(* IEC 61131-3 sources: ae-simplified-sorting-machine/AX/src/controlModules, 7 files *)

(* ---- IElevator.st ---- *)
NAMESPACE ControlModules

    /// Interface for elevator classes that extends ITransportDevice to add additional
    /// commands relevant for elevator operation
    INTERFACE IElevator extends ITransportDevice
        //=============================================================================
        //SIEMENS AG
        //(c)Copyright 2025 All Rights Reserved
        //-----------------------------------------------------------------------------
        //Tested with:   S7-1500 FW V4.0
        //Engineering:   SIMATIC AX Logic Control Engineering
        //Requirements:  none
        //Functionality: Interface for Transport Devices used as elevators
        //-----------------------------------------------------------------------------
        //Change log table:
        //Version  Date       Expert in charge                Changes applied
        //01.00.00 28.11.2025 Siemens Industry Online Support First Release
        //=============================================================================

        /// Commands the elevator to move upward continuously until upper limit is reached
        /// Enables movement without a specific target position
        METHOD  MoveUp
            VAR_INPUT
                /// Velocity for upward movement
                velocity : INT;
            END_VAR
        END_METHOD

        /// Commands the elevator to move downward continuously until lower limit is reached
        /// Enables movement without a specific target position
        METHOD  MoveDown
            VAR_INPUT
                /// Velocity for downward movement
                velocity : INT;
            END_VAR
        END_METHOD
    END_INTERFACE

END_NAMESPACE

(* ---- ITransportDevice.st ---- *)
NAMESPACE ControlModules

    /// Interface for Transport device Classes.
    INTERFACE ITransportDevice
        //=============================================================================
        //SIEMENS AG
        //(c)Copyright 2025 All Rights Reserved
        //-----------------------------------------------------------------------------
        //Tested with:   S7-1500 FW V4.0
        //Engineering:   SIMATIC AX Logic Control Engineering
        //Requirements:  none
        //Functionality: Interface used for control modules implemented as transport devices
        //-----------------------------------------------------------------------------
        //Change log table:
        //Version  Date       Expert in charge                Changes applied
        //01.00.00 28.11.2025 Siemens Industry Online Support First Release
        //=============================================================================

        /// Enables the transport device for operation
        /// Sets the internal enable flag to allow movement commands
        METHOD Enable
        END_METHOD

        /// Disables the transport device for operation
        /// Sets the internal enable flag to disable movement commands
        METHOD  Disable
        END_METHOD

        /// Stops the transport device operation
        /// Disables the device by setting the enable flag to FALSE
        METHOD  Stop
        END_METHOD

        /// Acknowledges errors on the transport device
        /// Sets the internal error acknowledgment flag to clear error conditions
        METHOD  AckError
        END_METHOD

        /// Gets the enable status of the transport device.
        /// TRUE if device is enabled, FALSE otherwise
        METHOD  GetIsEnabled : BOOL
        END_METHOD

        /// Gets the feedback status of the transport device.
        /// TRUE if movement is done, FALSE otherwise
        METHOD  GetIsDone : BOOL
        END_METHOD

        /// Gets the actual position of the transport device.
        /// Actual position in INT
        METHOD  GetActualPosition : INT
        END_METHOD

        /// Commands the transport device to move to a specified position.
        /// TRUE if movement command was accepted (device enabled), FALSE otherwise
        METHOD  PosAbsolute : BOOL
            VAR_INPUT
                /// Target position for the movement command
                targetPos : INT;
                /// Velocity for the movement (optional)
                velocity : INT := INT#0;
            END_VAR
        END_METHOD

        /// Moves the drive at a specified constant velocity.
        /// Sets the drive to jog mode and starts continuous movement.
        /// TRUE if movement command was accepted (device enabled), FALSE otherwise
        METHOD MoveVelocity : BOOL
            VAR_INPUT
                /// Velocity in LU (Length Units) for the drive
                velocity    : INT;
            END_VAR
        END_METHOD

        /// Executes a relative positioning movement.
        /// Moves the drive by a specified increment from current position.
        /// TRUE if movement command was accepted (device enabled), FALSE otherwise
        METHOD PosRelative : BOOL
            VAR_INPUT
                /// Position increment in LU to move relative to current position
                posIncrement   : INT;
                /// Velocity for the movement (uses last velocity if 0)
                velocity    : INT   := INT#0;
            END_VAR
        END_METHOD

        /// Retrieves the current status of the transport device.
        /// Status word containing device state information
        METHOD  GetStatus : WORD
        END_METHOD

        /// Gets if the transport device is in error state.
        /// TRUE if device is in error state, FALSE otherwise
        METHOD  GetIsError : BOOL
        END_METHOD

        /// Executes the transport device control logic.
        /// This method should be called cyclically in the main program loop.
        /// Abstract method that must be implemented by derived classes.
        METHOD Execute
        END_METHOD
    END_INTERFACE

END_NAMESPACE

(* ---- ConveyorSim.st ---- *)
USING System.Math;

NAMESPACE ControlModules

    /// Simulated conveyor class for transport operations without hardware dependency
    /// Extends TransportDevice to provide simulated drive control functionality
    /// Similar to ConveyorSinaPos but uses increment-based movement simulation like Elevator
    CLASS ConveyorSim
        EXTENDS TransportDevice
        //=============================================================================
        //SIEMENS AG
        //(c)Copyright 2025 All Rights Reserved
        //-----------------------------------------------------------------------------
        //Tested with:   S7-1500 FW V4.0
        //Engineering:   SIMATIC AX Logic Control Engineering
        //Requirements:  none
        //Functionality: Simulation of a conveyor control module
        //-----------------------------------------------------------------------------
        //Change log table:
        //Version  Date       Expert in charge                Changes applied
        //01.00.00 28.11.2025 Siemens Industry Online Support First Release
        //=============================================================================
        VAR PROTECTED
            /// Movement increment per execution cycle
            _cycleIncrement : INT := DEFAULT_CYCLE_INCREMENT;
            /// Stores last velocity for positioning commands
            _lastVelocity : INT := INT#0;
            /// Enable the movement simulation
            _moveEnable : BOOL := FALSE;
            /// Direction of movement for relative positioning
            _moveDirection : INT := INT#1; // 1 for positive, -1 for negative
            /// Target position for absolute positioning
            _targetPosition : INT := INT#0;
            /// Flag indicating if positioning is active
            _positioningActive : BOOL := FALSE;
            /// Mode of operation (similar to SinaPos modes)
            _operationMode : typeConveyorModuleMode := typeConveyorModuleMode#IDLE;
        END_VAR
        VAR CONSTANT
            /// Default cycle increment for movement simulation
            DEFAULT_CYCLE_INCREMENT : INT := INT#10;
        END_VAR
        /// Configures the simulated conveyor parameters
        METHOD PUBLIC SetConfig
            VAR_INPUT
                /// Movement increment per execution cycle (absolute value will be used)
                cycleIncrement : INT := INT#10;
            END_VAR
            _cycleIncrement := ABS(cycleIncrement);
        END_METHOD
        /// Stops the simulated conveyor and disables all commands
        /// Clears all pending commands and disables movement

        METHOD PUBLIC OVERRIDE Stop
            THIS.clearCommands();
        END_METHOD
        /// Moves the simulated drive at a specified constant velocity.
        /// Simulates continuous movement in positive direction.
        /// TRUE if movement command was accepted, FALSE otherwise
        METHOD PUBLIC OVERRIDE MoveVelocity : BOOL
            VAR_INPUT
                /// Velocity in LU (Length Units) for the drive (sign determines direction)
                velocity : INT;
            END_VAR
            // Clear possible remaining commands before triggering new commands
            THIS.clearCommands();
            // Set operation mode and parameters for velocity movement
            _operationMode := typeConveyorModuleMode#JOG;
            _lastVelocity := ABS(velocity); // Store absolute velocity
            // Determine direction based on velocity sign
            IF velocity >= 0 THEN
                _moveDirection := INT#1;
            ELSE
                _moveDirection := INT#-1;
            END_IF;
            // Set feedback variables
            _moveEnable := TRUE;
            _done := FALSE;
            MoveVelocity := _moveEnable;
        END_METHOD
        /// Executes a relative positioning movement.
        /// Moves the drive by a specified increment from current position.
        /// TRUE if movement command was accepted, FALSE otherwise
        METHOD PUBLIC OVERRIDE PosRelative : BOOL
            VAR_INPUT
                /// Position increment in LU to move relative to current position
                posIncrement : INT;
                /// Velocity for the movement (uses last velocity if 0)
                velocity : INT := INT#0;
            END_VAR
            // Clear actual commands before starting new command
            THIS.clearCommands();
            // Use velocity input in case a velocity is given
            IF velocity <> INT#0 THEN
                _lastVelocity := ABS(velocity);
            END_IF;
            // Set parameters for relative positioning
            _operationMode := typeConveyorModuleMode#RELATIVE_POSITIONING;
            _targetPosition := _actualPos + posIncrement;
            // Determine direction based on increment sign
            IF posIncrement >= 0 THEN
                _moveDirection := INT#1;
            ELSE
                _moveDirection := INT#-1;
            END_IF;
            // Set feedback variables
            _positioningActive := TRUE;
            _moveEnable := TRUE;
            _done := FALSE;
            PosRelative := _moveEnable;
        END_METHOD

        /// Executes an absolute positioning movement.
        /// Moves the drive to a specified absolute position.
        /// TRUE if movement command was accepted, FALSE otherwise
        METHOD PUBLIC OVERRIDE PosAbsolute : BOOL
            VAR_INPUT
                /// Target position for the movement
                targetPos : INT;
                /// Velocity for the movement (optional)
                velocity : INT := INT#0;
            END_VAR
            // Clear actual commands before starting new command
            THIS.clearCommands();
            // Set parameters for absolute positioning
            _operationMode := typeConveyorModuleMode#ABSOLUTE_POSITIONING;
            _targetPosition := targetPos;
            // Determine direction based on target vs current position
            IF targetPos >= _actualPos THEN
                _moveDirection := INT#1;
            ELSE
                _moveDirection := INT#-1;
            END_IF;
            // Use velocity input in case a velocity is given
            IF velocity <> INT#0 THEN
                _lastVelocity := ABS(velocity);
            END_IF;
            _positioningActive := TRUE;
            _moveEnable := TRUE;
            _done := FALSE;
            PosAbsolute := TRUE;
        END_METHOD

        /// Sets the current position as the home/reference position
        /// Simulates homing by setting current position to zero
        METHOD PUBLIC SetHomePosition
            THIS.clearCommands();
            _actualPos := INT#0;
            _operationMode := typeConveyorModuleMode#SET_HOME_POSITION;
        END_METHOD

        /// Checks if the drive axis has been referenced/homed.
        /// For simulation, always returns TRUE as homing is instant.
        /// TRUE (always referenced in simulation)
        METHOD PUBLIC IsHomed : BOOL
            IsHomed := TRUE; // Always homed in simulation
        END_METHOD

        /// Gets the completion status of positioning operations.
        /// TRUE if positioning operation is completed, FALSE if still moving
        METHOD PUBLIC OVERRIDE GetIsDone : BOOL
            GetIsDone := _done;
        END_METHOD

        /// Clears all active commands and resets drive parameters
        /// Used internally when starting a new command to prevent conflicts
        METHOD PROTECTED clearCommands
            _moveEnable := FALSE;
            _positioningActive := FALSE;
            _operationMode := typeConveyorModuleMode#IDLE;
            _moveDirection := INT#1;
        END_METHOD

        /// Executes the simulated conveyor control logic cyclically
        /// Simulates movement by incrementing position values
        /// This method should be called in every cycle of the main program
        METHOD PUBLIC OVERRIDE Execute
            VAR_TEMP
                increment : INT := INT#0;
                positionDifference : INT := INT#0;
            END_VAR
            // Handle error acknowledgment
            IF _ackError THEN
                _error := FALSE;
                _status := typeTransportDeviceBaseStatus#STATUS_NO_CALL;
                _ackError := FALSE;
            END_IF;
            // Only move if enabled and movement is active
            IF _enable AND _moveEnable AND NOT _error THEN
                CASE _operationMode OF
                    typeConveyorModuleMode#IDLE:
                        // Idle mode - no movement
                        _status := typeTransportDeviceBaseStatus#STATUS_IDLE;
                        _done := TRUE;
                        _moveEnable := FALSE;
                    typeConveyorModuleMode#JOG:
                        // Continuous movement based on velocity
                        increment := _moveDirection * _cycleIncrement;
                        _actualPos := _actualPos + increment;
                        _done := FALSE; // Jog mode never completes
                        _status := typeTransportDeviceBaseStatus#STATUS_MOVING;
                    typeConveyorModuleMode#RELATIVE_POSITIONING, typeConveyorModuleMode#ABSOLUTE_POSITIONING:
                        // Positioning movement towards target
                        IF _positioningActive THEN
                            positionDifference := _targetPosition - _actualPos;
                            _status := typeTransportDeviceBaseStatus#STATUS_POSITIONING;
                            // Check if target is reached
                            IF ABS(positionDifference) <= _cycleIncrement THEN
                                // Target reached - set exact position and stop
                                _actualPos := _targetPosition;
                                _moveEnable := FALSE;
                                _positioningActive := FALSE;
                                _done := TRUE;
                                _operationMode := typeConveyorModuleMode#IDLE;
                            ELSE
                                // Continue moving towards target
                                increment := _moveDirection * _cycleIncrement;
                                _actualPos := _actualPos + increment;
                                _done := FALSE;
                            END_IF;
                        END_IF;
                    typeConveyorModuleMode#SET_HOME_POSITION:
                        // Home position setting is instant in simulation
                        _operationMode := typeConveyorModuleMode#IDLE;
                        _done := TRUE;
                END_CASE;
            ELSE
                // Not enabled or error - ensure stopped state
                _moveEnable := FALSE;
                _positioningActive := FALSE;
            END_IF;
        END_METHOD
    END_CLASS

END_NAMESPACE

(* ---- ConveyorSinaPos.st ---- *)
USING Simatic.Ax.Sinamics;

NAMESPACE ControlModules

    /// Class for controlling a SinaPos control module as a transport device
    /// Extends TransportDevice to provide Sinamics drive control functionality
    CLASS ConveyorSinaPos EXTENDS TransportDevice
        //=============================================================================
        //SIEMENS AG
        //(c)Copyright 2025 All Rights Reserved
        //-----------------------------------------------------------------------------
        //Tested with:   S7-1500 FW V4.0
        //Engineering:   SIMATIC AX Logic Control Engineering
        //Requirements:  none
        //Functionality: Conveyor control with Sinamics drive using SinaPos telegram
        //-----------------------------------------------------------------------------
        //Change log table:
        //Version  Date       Expert in charge                Changes applied
        //01.00.00 28.11.2025 Siemens Industry Online Support First Release
        //=============================================================================
        VAR PROTECTED
            _sinaPosDrive   : SinaPos;              // Sina Pos FB call to control the drive
            _lastVelocity   : INT       := INT#0;   // Stores last velocity for positioning commands
        END_VAR

        /// Configures the SinaPos drive parameters and hardware connections
        METHOD PUBLIC SetConfigSina
            VAR_INPUT
                /// Configuration for axis parameters
                configSinaPos : SinaPosConfiguration;
                /// Hardware ID of the SIMATIC S7-1200/1500 setpoint slot
                hwidSTW : UINT;
                /// Hardware ID of the SIMATIC S7-1200/1500 actual value slot
                hwidZSW : UINT;
                /// Set Sina Pos mode of operation
                mode : SinaPosMode;
            END_VAR
            _sinaPosDrive.config := configSinaPos;
            _sinaPosDrive.hwidSTW := hwidSTW;
            _sinaPosDrive.hwidZSW := hwidZSW;
            _sinaPosDrive.mode := mode;
        END_METHOD

        /// Stops the SinaPos drive and disables all commands
        /// Clears all pending commands and disables the drive
        METHOD PUBLIC OVERRIDE Stop
            THIS.clearCommands();
            _enable := FALSE;
        END_METHOD

        /// Moves the drive at a specified constant velocity.
        /// Sets the drive to jog mode and starts continuous movement.
        /// TRUE if movement command was accepted, FALSE otherwise
        METHOD PUBLIC OVERRIDE MoveVelocity : BOOL
            VAR_INPUT
                /// Velocity for the movement
                velocity    : INT;
            END_VAR
            // Clear possible remaining commands befor triggering new commands
            THIS.clearCommands();
            // Set Velocity and jog mode to run as Move velocity
            _sinaPosDrive.mode := SinaPosMode#Jog;
            _sinaPosDrive.velocity := velocity;
            _sinaPosDrive.jog1 := TRUE;
            MoveVelocity := TRUE;
        END_METHOD

        /// Executes a relative positioning movement.
        /// Moves the drive by a specified increment from current position.
        /// TRUE if movement command was accepted, FALSE otherwise
        METHOD PUBLIC OVERRIDE PosRelative : BOOL
            VAR_INPUT
                /// Position increment in LU to move relative to current position
                posIncrement   : INT;
                /// Velocity for the movement (uses last velocity if 0)
                velocity    : INT   := INT#0;
            END_VAR
            // Clear actual commands before starting new command
            THIS.clearCommands();
            // Use velocity input incase no velocity is given
            IF (NOT (velocity = INT#0)) THEN
                _lastVelocity := velocity;
            END_IF;
            // Set Sina pos parameters for relative positioning
            _sinaPosDrive.mode := SinaPosMode#RelativePositioning;
            _sinaPosDrive.position := posIncrement;
            _sinaPosDrive.velocity := _lastVelocity;
            _sinaPosDrive.executeMode := TRUE;
            PosRelative := TRUE;
        END_METHOD

        /// Executes an absolute positioning movement.
        /// Moves the drive to a specified absolute position.
        /// TRUE if movement command was accepted, FALSE otherwise
        METHOD PUBLIC OVERRIDE PosAbsolute : BOOL
            VAR_INPUT
                /// Target position for the movement
                targetPos : INT;
                /// Velocity for the movement (optional)
                velocity : INT := INT#0;
            END_VAR
            // Clear actual commands before starting new command
            THIS.clearCommands();
            // Use velocity input incase no velocity is given
            IF (NOT (velocity = INT#0)) THEN
                _lastVelocity := velocity;
            END_IF;
            // Set Sina pos parameters for relative positioning
            _sinaPosDrive.mode := SinaPosMode#AbsolutePositioning;
            _sinaPosDrive.position := targetPos;
            _sinaPosDrive.velocity := _lastVelocity;
            _sinaPosDrive.executeMode := TRUE;
            PosAbsolute := TRUE;
        END_METHOD

        /// Sets the current position as the home/reference position
        /// Establishes the current drive position as the zero reference point
        METHOD PUBLIC SetHomePosition
            THIS.clearCommands();
            _sinaPosDrive.mode := SinaPosMode#SetHomePosition;
            _sinaPosDrive.executeMode := TRUE;
        END_METHOD

        /// Checks if the drive axis has been referenced/homed.
        /// Returns TRUE if axis is referenced and ready for positioning, FALSE otherwise
        METHOD PUBLIC IsHomed : BOOL
            IsHomed := _sinaPosDrive.axisReferenced;
        END_METHOD

        /// Clears all active commands and resets drive parameters
        /// Used internally when starting a new command to prevent conflicts
        METHOD PROTECTED clearCommands
            _sinaPosDrive.position := INT#0;
            _sinaPosDrive.jog1 := FALSE;
            _sinaPosDrive.jog2 := FALSE;
            _sinaPosDrive.executeMode := FALSE;
        END_METHOD

        /// Executes the SinaPos drive control logic cyclically
        /// Calls the SinaPos function block and updates status information
        /// This method should be called in every cycle of the main program
        METHOD PUBLIC OVERRIDE Execute
            // Call Sina Pos FB for Drive control and feedback
            _sinaPosDrive(
                enableAxis := _enable,
                AcknowledgeError := _ackError,
                error => _error,
                status => _status,
                axisPositionOk => _done
                );
            // Get feedback from Drive call
            _actualPos := TO_INT(_sinaPosDrive.actualPosition); // Sina Pos gets the Value in DINT with LU units
            // Reset acknowledge error flag after processing
            IF _ackError AND  NOT _sinaPosDrive.error THEN
                _ackError := FALSE;
                _status := typeTransportDeviceBaseStatus#STATUS_NO_CALL;
            END_IF;
            IF _done THEN
                THIS.clearCommands();
            END_IF;
        END_METHOD
    END_CLASS
END_NAMESPACE

(* ---- ElevatorSim.st ---- *)
USING System.Math;

NAMESPACE ControlModules

    /// Elevator class for vertical transport operations
    /// Extends TransportDevice to provide elevator-specific functionality for material handling
    CLASS ElevatorSim EXTENDS TransportDevice IMPLEMENTS IElevator
        //=============================================================================
        //SIEMENS AG
        //(c)Copyright 2025 All Rights Reserved
        //-----------------------------------------------------------------------------
        //Tested with:   S7-1500 FW V4.0
        //Engineering:   SIMATIC AX Logic Control Engineering
        //Requirements:  none
        //Functionality: Simulation of an elevator control module
        //-----------------------------------------------------------------------------
        //Change log table:
        //Version  Date       Expert in charge                Changes applied
        //01.00.00 28.11.2025 Siemens Industry Online Support First Release
        //=============================================================================
        VAR PROTECTED
            /// Move positioning increment for each execute call
            _cycleIncrement : INT  := INT#10;
            /// Max upper value for actual position
            _upperLimit : INT  := INT#100;
            /// Min lower value for actual position
            _lowerLimit : INT  := INT#0;
            /// Direction of movement. TRUE for up and FALSE for down
            _direction : BOOL  := TRUE;
            /// Enable the Movement
            _moveEnable : BOOL  := FALSE;
            /// Movement without target enabled
            _moveUntilLimit : BOOL  := FALSE;
        END_VAR
        VAR CONSTANT
            DIRECTION_UP : BOOL  := TRUE;
            DIRECTION_DOWN : BOOL  := FALSE;
        END_VAR

        /// Configures the elevator movement parameters and position limits
        METHOD PUBLIC SetConfigLimits
            VAR_INPUT
                /// Movement increment per execution cycle (absolute value will be used)
                cycleIncrement : INT;
                /// Maximum allowed position for elevator movement
                upperLimit : INT;
                /// Minimum allowed position for elevator movement
                lowerLimit : INT;
            END_VAR
            // Take Absolute value of increment
            _cycleIncrement := ABS(cycleIncrement);
            _upperLimit := upperLimit;
            _lowerLimit := lowerLimit;
            _actualPos := lowerLimit;
        END_METHOD

        /// Returns the inverted elevator position for HMI display (0 = up, 100 = down)
        /// Due to specific assembly crane SVG requirements
        METHOD PUBLIC GetInvertedPosition : INT
            GetInvertedPosition := 100 - _actualPos;
        END_METHOD

        /// Commands the elevator to move upward continuously until upper limit is reached
        /// Enables movement without a specific target position
        METHOD PUBLIC MoveUp
            VAR_INPUT
                /// Velocity for upward movement (optional, uses current if 0)
                velocity : INT;
            END_VAR
            // Enable movement witout target
            _moveUntilLimit := TRUE;
            _direction := DIRECTION_UP;
            _moveEnable := TRUE;
            // Set velocity if value given
            IF NOT (velocity = INT#0) THEN
                _cycleIncrement := velocity;
            END_IF;
        END_METHOD

        /// Commands the elevator to move downward continuously until lower limit is reached
        /// Enables movement without a specific target position
        METHOD PUBLIC MoveDown
            VAR_INPUT
                /// Velocity for downward movement (optional, uses current if 0)
                velocity : INT;
            END_VAR
            // Enable movement witout target
            _moveUntilLimit := TRUE;
            _direction := DIRECTION_DOWN;
            _moveEnable := TRUE;
            // Set velocity if value given
            IF NOT (velocity = INT#0) THEN
                _cycleIncrement := velocity;
            END_IF;
        END_METHOD

        /// Stops all elevator movement operations
        /// Disables both targeted and continuous movement modes
        METHOD PUBLIC OVERRIDE Stop
            _moveUntilLimit := FALSE;
            _moveEnable := FALSE;
        END_METHOD

        /// Commands the elevator to move to a specific target position.
        /// Validates target position against configured limits and determines movement direction.
        /// TRUE if movement command was accepted, FALSE if target is out of limits or error occurred
        METHOD PUBLIC  OVERRIDE PosAbsolute : BOOL
            VAR_INPUT
                /// Target position for the elevator movement
                targetPos : INT;
                /// Velocity for downward movement (optional, uses current if 0)
                velocity : INT := INT#0;
            END_VAR
            // Disable movement without target if active
            _moveUntilLimit := FALSE;
            // Define return value if operation not accepted
            PosAbsolute := FALSE;
            // If target position is outide of limits, trigger error.
            IF (targetPos < _lowerLimit) OR (targetPos > _upperLimit) THEN
                _error := TRUE;
                _status := typeTransportDeviceBaseStatus#ERR_TARGET_OUT_OF_LIMITS;
                RETURN;
            END_IF;
            // Set cycle increment velocity if velocity is unequal 0
            IF (velocity <> INT#0) THEN
                _cycleIncrement := velocity;
            END_IF;
            // Update target position
            _targetPos := targetPos;
            // Get the direction to move to
            IF _actualPos < _targetPos THEN
                _direction := DIRECTION_UP;
            ELSIF _actualPos > _targetPos THEN
                _direction := DIRECTION_DOWN;
            ELSE
                // Already at target, no movement needed
                _moveEnable := FALSE;
                _done := TRUE;
                RETURN;
            END_IF;
            // Enable flag for movement
            _moveEnable := TRUE;
            _done := FALSE;
            PosAbsolute := TRUE;
        END_METHOD

        /// Executes the elevator control logic cyclically
        /// Handles position updates, target reaching detection, and limit enforcement
        /// This method should be called in every cycle of the main program
        METHOD PUBLIC OVERRIDE Execute
            VAR_TEMP
                /// Position increment for every cycle
                increment : INT := INT#0;
            END_VAR
            /// Resets pending error.
            IF _ackError THEN
                _error := FALSE;
                _status := typeTransportDeviceBaseStatus#STATUS_NO_CALL;
                _ackError := FALSE;
            END_IF;

            // Exit if module not enabled to run
            IF NOT (_enable AND _moveEnable AND NOT _error) THEN
                RETURN;
            END_IF;
            // Cycle increment direction adaption
            IF _direction = DIRECTION_UP THEN
                // Direction up, increment positive
                increment := _cycleIncrement;
            ELSE
                // Direction down, increment negative
                increment := - _cycleIncrement;
            END_IF;
            // Update the actual position adding the cycle increment
            _actualPos := _actualPos + increment;
            // Mode with Target is active
            IF NOT _moveUntilLimit THEN
                // If the target is reached OR it over/under shoot the value, set actual position
                // as target position and stop movement
                IF (_actualPos = _targetPos)
                    OR (_direction = DIRECTION_UP AND _actualPos > _targetPos)
                    OR (_direction = DIRECTION_DOWN AND _actualPos < _targetPos) THEN
                    _actualPos := _targetPos;
                    _moveEnable := FALSE;
                    _done := TRUE;
                ELSE
                    _done := FALSE;
                END_IF;
            END_IF;
            // Get if Elevator is over the limit because of the cycle increment
            IF _actualPos > _upperLimit THEN
                _actualPos := _upperLimit;
                _moveEnable := FALSE;
            ELSIF _actualPos < _lowerLimit THEN
                _actualPos := _lowerLimit;
                _moveEnable := FALSE;
            END_IF;
        END_METHOD
    END_CLASS
END_NAMESPACE

(* ---- ElevatorSinaSpeedSim.st ---- *)
USING Simatic.Ax.Sinamics;

NAMESPACE ControlModules

    CLASS ElevatorSinaSpeedSim EXTENDS ElevatorSim
        //=============================================================================
        //SIEMENS AG
        //(c)Copyright 2025 All Rights Reserved
        //-----------------------------------------------------------------------------
        //Tested with:   S7-1500 FW V4.0
        //Engineering:   SIMATIC AX Logic Control Engineering
        //Requirements:  none
        //Functionality: Elevator control with Sinamics drive using SinaSpeed telegram
        //-----------------------------------------------------------------------------
        //Change log table:
        //Version  Date       Expert in charge                Changes applied
        //01.00.00 28.11.2025 Siemens Industry Online Support First Release
        //=============================================================================
        VAR PROTECTED
            /// Controller for Sina Speed supported telegrams
            _sinaSpeedDrive : SinaSpeed;
            /// Default Speed when none is given
            _defaultVelocity : INT;
        END_VAR
        /// Configures the SinaSpeed drive parameters and elevator limits
        METHOD PUBLIC SetConfigSina
            VAR_INPUT
                /// Configuration for SinaSpeed axis parameters
                sinaSpeedConfig : SinaSpeedConfiguration;
                /// Reference speed for the drive in engineering units
                sinaRefSpeed : REAL;
                /// Default velocity for the elevator
                defaultVelocity : INT;
                /// Hardware ID of the SIMATIC S7-1200/1500 setpoint slot
                hwidSTW : UINT;
                /// Hardware ID of the SIMATIC S7-1200/1500 actual value slot
                hwidZSW : UINT;
            END_VAR
            // Set sina settings
            _sinaSpeedDrive.config := sinaSpeedConfig;
            _sinaSpeedDrive.referenceSpeed := sinaRefSpeed;
            _sinaSpeedDrive.hwidSTW := hwidSTW;
            _sinaSpeedDrive.hwidZSW := hwidZSW;
            _defaultVelocity := defaultVelocity;
        END_METHOD

        METHOD PUBLIC OVERRIDE Execute
            // Call SinaSpeed control to write and read data
            _sinaSpeedDrive(enableAxis := _enable AND _moveEnable, acknowledgeError :=  _ackError,
            error => _error, status => _status);
            SUPER.Execute();
        END_METHOD

        METHOD PUBLIC OVERRIDE Disable
            SUPER.Disable();
            // Call SinaSpeed control to write and read data
            _sinaSpeedDrive(enableAxis := _enable AND _moveEnable, acknowledgeError :=  _ackError,
            error => _error, status => _status);
        END_METHOD

        /// Commands the elevator to move upward continuously until upper limit is reached
        /// Enables movement without a specific target position
        METHOD PUBLIC OVERRIDE MoveUp
            VAR_INPUT
                /// Velocity for upward movement (absolute value will be used)
                velocity : INT;
            END_VAR
            VAR_TEMP
                velocityValue : INT;
            END_VAR
            // Do not move Up when at upper limit
            IF _actualPos >= _upperLimit THEN // TODO: error/warning? also in the super?
                RETURN;
            END_IF;
            // Set velocity for MoveVelocity with default or input velocity
            IF velocity = INT#0 THEN
                velocityValue := _defaultVelocity;
            ELSE
                velocityValue := System.Math.Abs(velocity);
            END_IF;
            // Call base method to handle most configuration
            SUPER.MoveUp();
            // Enable movement without target
            THIS.MoveVelocity(velocityValue);
        END_METHOD

        /// Commands the elevator to move downward continuously until lower limit is reached
        /// Enables movement without a specific target position
        METHOD PUBLIC OVERRIDE MoveDown
            VAR_INPUT
                /// Velocity for downward movement (absolute value will be used)
                velocity : INT;
            END_VAR
            VAR_TEMP
                velocityValue : INT;
            END_VAR
            // Do not move Down when at lower limit
            IF _actualPos <= _lowerLimit THEN // TODO: error/warning? also in the super?
                RETURN;
            END_IF;
            // Set velocity for MoveVelocity with default ot input velocity
            IF velocity = INT#0 THEN
                velocityValue := - _defaultVelocity;
            ELSE
                velocityValue := - System.Math.Abs(velocity);
            END_IF;
            // Call base mathod to handle most configuration
            SUPER.MoveDown();
            // Enable movement witout target
            THIS.MoveVelocity(velocityValue);
        END_METHOD

        METHOD PUBLIC OVERRIDE MoveVelocity : BOOL
            VAR_INPUT
                velocity : INT;
            END_VAR
            // Ge movement direction
            IF velocity >= INT#0 THEN
                _direction := DIRECTION_UP;
            ELSE
                _direction := DIRECTION_DOWN;
            END_IF;
            // Enable movement witout target
            _moveUntilLimit := TRUE;
            _moveEnable := TRUE;
            // Set speed to sina speed block
            _sinaSpeedDrive.speedSetpoint := velocity;
            MoveVelocity := TRUE;
        END_METHOD

        /// Get Diagnostics ID from Sina Speed for troubleshooting
        METHOD PUBLIC GetDiagId : WORD
            GetDiagId := _sinaSpeedDrive.diagnosticsId;
        END_METHOD
    END_CLASS
END_NAMESPACE

(* ---- TransportDevice.st ---- *)
NAMESPACE ControlModules
    /// Transport device class for controlling movement and positioning
    /// Used in sorting machine applications to handle material transport
    CLASS ABSTRACT TransportDevice IMPLEMENTS ITransportDevice
        //=============================================================================
        //SIEMENS AG
        //(c)Copyright 2025 All Rights Reserved
        //-----------------------------------------------------------------------------
        //Tested with:   S7-1500 FW V4.0
        //Engineering:   SIMATIC AX Logic Control Engineering
        //Requirements:  none
        //Functionality: Basis abstract class for transport device control modules
        //-----------------------------------------------------------------------------
        //Change log table:
        //Version  Date       Expert in charge                Changes applied
        //01.00.00 28.11.2025 Siemens Industry Online Support First Release
        //=============================================================================
        VAR PROTECTED
            /// Enable flag for device operation
            _enable : BOOL := FALSE;
            /// Feedback flag for movement done
            _done : BOOL := FALSE;
            /// Current actual position of the transport device
            _actualPos : INT := INT#0;
            /// Target position for movement commands
            _targetPos : INT := INT#0;
            /// Error flag indicating device fault state
            _error : BOOL := FALSE;
            /// Acknowkledge Error during Execute
            _ackError : BOOL := FALSE;
            /// Status word containing device state information
            _status : typeTransportDeviceBaseStatus;
        END_VAR
        /// Enables the transport device for operation
        /// Sets the internal enable flag to allow movement commands
        METHOD PUBLIC Enable
            _enable := TRUE;
        END_METHOD

        /// Disables the transport device for operation
        /// Sets the internal enable flag to disable movement commands
        METHOD PUBLIC Disable
            _enable := FALSE;
            _done := FALSE;
        END_METHOD

        /// Stops the transport device operation
        /// Disables the device by setting the enable flag to FALSE
        METHOD PUBLIC Stop
            _enable := FALSE;
            _done := FALSE;
        END_METHOD

        /// Acknowledges errors on the transport device
        /// Sets the internal error acknowledgment flag to clear error conditions
        METHOD PUBLIC AckError
            _ackError := TRUE;
        END_METHOD

        /// Gets the enable status of the transport device
        METHOD PUBLIC GetIsEnabled : BOOL
            GetIsEnabled := _enable;
        END_METHOD

        /// Gets the feedback status of the transport device.
        /// TRUE if movement is done, FALSE otherwise
        METHOD PUBLIC GetIsDone : BOOL
            GetIsDone := _done;
        END_METHOD

        /// Gets the actual position of the transport device
        METHOD PUBLIC GetActualPosition : INT
            GetActualPosition := _actualPos;
        END_METHOD

        /// Commands the transport device to move to a specified position (not supported in base class)
        /// Return FALSE if not supported
        METHOD PUBLIC PosAbsolute : BOOL
            VAR_INPUT
                /// Target position for the movement command
                targetPos : INT;
                /// Velocity for the movement (optional)
                velocity : INT := INT#0;
            END_VAR
            _status := typeTransportDeviceBaseStatus#ERR_COMMAND_NOT_SUPPORTED;
            _error := TRUE;
            PosAbsolute := FALSE;
        END_METHOD

        /// Moves the drive at a specified constant velocity (not supported in base class)
        /// Return FALSE if not supported
        METHOD PUBLIC MoveVelocity : BOOL
            VAR_INPUT
                /// Velocity in LU (Length Units) for the drive
                velocity : INT;
            END_VAR
            _status := typeTransportDeviceBaseStatus#ERR_COMMAND_NOT_SUPPORTED;
            _error := TRUE;
            MoveVelocity := FALSE;
         END_METHOD

        /// Executes a relative positioning movement (not supported in base class)
        /// Return FALSE if not supported
        METHOD PUBLIC PosRelative : BOOL
            VAR_INPUT
                /// Position increment in LU to move relative to current position
                posIncrement : INT;
                /// Velocity for the movement (uses last velocity if 0)
                velocity : INT := INT#0;
            END_VAR
            _status := typeTransportDeviceBaseStatus#ERR_COMMAND_NOT_SUPPORTED;
            _error := TRUE;
            PosRelative := FALSE;
         END_METHOD

        /// Retrieves the current status of the transport device
        METHOD PUBLIC GetStatus : WORD
            GetStatus := _status;
        END_METHOD

        /// Get is the transport device in error state
        METHOD PUBLIC GetIsError : BOOL
            GetIsError := _error;
        END_METHOD

        /// Executes the transport device control logic
        /// This method should be called cyclically in the main program loop
        /// Abstract method that must be implemented by derived classes
        METHOD PUBLIC ABSTRACT Execute
        END_METHOD

    END_CLASS

END_NAMESPACE
